FUNCTION_BLOCK E_TABLE (* Composite Function Block Type *)
  (* Standard: 61499-1 Annex A; Description: Copyright (c) 2017 fortiss GmbH This program and the accompanying materials are made available under the terms of the Eclipse Public License 2.0 which is available at https://www.eclipse.org/legal/epl-2.0/ SPDX-License-Identifier: EPL-2.0 *)
  (* Version 1.0, 2017-09-22, Alois Zoitl, fortiss GmbH, initial API and implementation and/or initial documentation *)
  (* Version 3.0, 2025-04-14, Patrick Aigner, changed package *)
  PACKAGE iec61499::events;
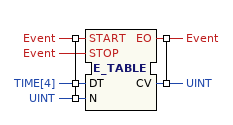
  EVENT_INPUT
    START WITH DT, N; (* Start table driven event generation *)
    STOP; (* Stop table driven event generation *)
  END_EVENT
  EVENT_OUTPUT
    EO WITH CV; (* Generated events: N events at periods DT, starting at DT[0] after START *)
  END_EVENT
  VAR_INPUT
    DT : ARRAY [0..3] OF TIME; (* Periods between events *)
    N : UINT; (* Number of events to generate *)
  END_VAR
  VAR_OUTPUT
    CV : UINT; (* Current event index, 0..N-1 *)
  END_VAR
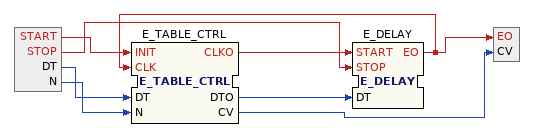
  FBS
    E_TABLE_CTRL : iec61499::events::E_TABLE_CTRL;
    E_DELAY : iec61499::events::E_DELAY;
  END_FBS
  EVENT_CONNECTIONS
    E_TABLE_CTRL.CLKO TO E_DELAY.START;
    E_DELAY.EO TO EO;
    START TO E_TABLE_CTRL.INIT;
    E_DELAY.EO TO E_TABLE_CTRL.CLK;
    STOP TO E_DELAY.STOP;
  END_CONNECTIONS
  DATA_CONNECTIONS
    E_TABLE_CTRL.DTO TO E_DELAY.DT;
    E_TABLE_CTRL.CV TO CV;
    DT TO E_TABLE_CTRL.DT;
    N TO E_TABLE_CTRL.N;
  END_CONNECTIONS
END_FUNCTION_BLOCK
